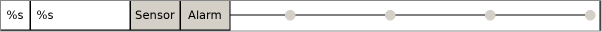
VISUALIZATION V_LiquidSensorState  // 602x32
VAR_IN_OUT
	IOfbLiquidSensor : FB_LiquidSensor;
END_VAR
    Line (590,15) (230,15), colour toggle: IOfbLiquidSensor.QbLMStatus, invisible if: IOfbLiquidSensor.VnvdwCFGLiquidToTransor.4 = 0
    Ellipse (585,10 10x10), colour toggle: IOfbLiquidSensor.QbLMStatus, invisible if: IOfbLiquidSensor.VnvdwCFGLiquidToTransor.4 = 0
    Line (490,15) (230,15), colour toggle: IOfbLiquidSensor.QbLMStatus, invisible if: IOfbLiquidSensor.VnvdwCFGLiquidToTransor.3 = 0
    Ellipse (485,10 10x10), colour toggle: IOfbLiquidSensor.QbLMStatus, invisible if: IOfbLiquidSensor.VnvdwCFGLiquidToTransor.3 = 0
    Line (390,15) (230,15), colour toggle: IOfbLiquidSensor.QbLMStatus, invisible if: IOfbLiquidSensor.VnvdwCFGLiquidToTransor.2 = 0
    Ellipse (385,10 10x10), colour toggle: IOfbLiquidSensor.QbLMStatus, invisible if: IOfbLiquidSensor.VnvdwCFGLiquidToTransor.2 = 0
    Rectangle (0,0 30x30), "%s", text variable: IOfbLiquidSensor.iChan
    Rectangle (30,0 100x30), "%s", text variable: IOfbLiquidSensor.VnvszName
    Rectangle (180,0 50x30), "Alarm", colour toggle: IOfbLiquidSensor.QbLMStatus
    Line (290,15) (230,15), colour toggle: IOfbLiquidSensor.QbLMStatus, invisible if: IOfbLiquidSensor.VnvdwCFGLiquidToTransor.1 = 0
    Ellipse (285,10 10x10), colour toggle: IOfbLiquidSensor.QbLMStatus, invisible if: IOfbLiquidSensor.VnvdwCFGLiquidToTransor.1 = 0
    Line (600,30) (600,0)
    Rectangle (130,0 50x30), "Sensor", colour toggle: IOfbLiquidSensor.IbLiquidSensor
END_VISUALIZATION

(* stored: Version 1.1.0.1, ProductVersion 3.1.4018.10
   Visu V_LiquidSensorState: Id {ac2f2fc4-edaf-489b-a301-58efa8dfcfd6} *)
